// TIA Portal V19 export
TYPE "LAF_typeMemCardDiag"
TITLE = Siemens Memory Card diagnostic / Siemens Memory Card Diagnose
// Type contains the information that is displayed in the visualization. / SMC Diagnose
// stored: Access Published
   STRUCT
      alarmWarnInfo : Byte;   // Alarms/Warnings/Information: %X0:AM1, %X1:AM2, %X2:AM3, %X3:AM4, %X4:WM5, %X5:AM6, %X6:WM7, %X7:IM8 / Störungen/Warnungen/Informationen: %X0:AM1, %X1:AM2, %X2:AM3, %X3:AM4, %X4:WM5, %X5:AM6, %X6:WM7, %X7:IM8
      manualUpdate : Bool;   // Manueller Update der Informationen / Manual update of the information
      memorySpaceKbyte : UDInt;   // Memory size in KB (1 KB = 1024 bytes) / Speichergröße in KByte (1 KByte = 1024 Byte)
      assignedMemorySpaceKbyte : UDInt;   // Assigned memory space in KB / Belegter Speicherplatz in KByte
      assignedMemorySpace : UDInt;   // Assigned memory space in % / Belegter Speicherplatz in %
      usedLifetime : UDInt;   // Maintenance information: Previously used up portion of the service life in % / Wartungsinformation: Bisher verbrauchter Anteil der Lebensdauer in %
      paraLifetime : UDInt;   // Set proportion of the service life as a percentage after which the CPU creates a diagnostics buffer entry and activates the maintenance LED / Parametrierter Anteil der Lebensdauer in %, nach dessen Ablauf die CPU einen Diagnosepuffereintrag erstellt und die Maintenance-LED einschaltet
      warningFromMemorySpace : UDInt := 81;   // Warning from Assigned Memory Space (in %) / Warnung auslösen ab belegtem Speicherplatz (in %)
      alarmFromMemorySpace : UDInt := 95;   // Alarm from Assigned Memory Space (in %) / Alarm auslösen ab belegtem Speicherplatz (in %)
   END_STRUCT;
END_TYPE
